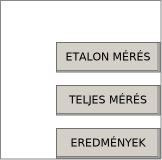
VISUALIZATION Vegmero_teljes  // 162x160
    Button (56,85 104x30), "TELJES MÉRÉS", input disabled if: VEGMERO.s_InCommand<>''
        OnMouseUp: execute { VEGMERO.s_InCommand:='TELJESMERES'; GVL.bMeresiEredmenyekRejtve:=FALSE; }
    Button (56,128 104x30), "EREDMÉNYEK"
        OnMouseUp: execute { GVL.bMeresiEredmenyekRejtve:=FALSE; }
    Button (56,42 104x30), "ETALON MÉRÉS", input disabled if: VEGMERO.s_InCommand<>''
        OnMouseUp: execute { VEGMERO.s_InCommand:='ETALONMERES'; GVL.bMeresiEredmenyekRejtve:=FALSE; }
END_VISUALIZATION

(* stored: Version 1.1.0.1, ProductVersion 3.1.4024.11
   Visu Vegmero_teljes: Id {eaa770f4-ede0-49d7-a878-85b3bc9cb285} *)
